Staubli VAL3: cycle_isRun.pgx

program cycle_isRun(bool& x_bStatus[] (dimensions=1))
begin
  //
  // ask for the cycle running
  //
  x_bStatus=cycleStatus:bCycle
end
